Omron CX-Programmer project 新規ﾌﾟﾛｼﾞｪｸﾄ (CX-Programmer 9.61)

# PLC hoge1: CP1L L

## Program 新規ﾌﾟﾛｸﾞﾗﾑ1 (cyclic task 0)
Local symbols
I 0.00 BOOL
Q 100.00 BOOL

### Section ｾｸｼｮﾝ1

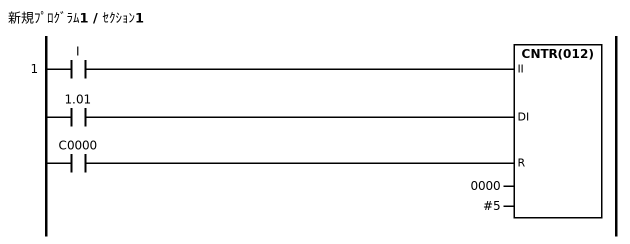
; rung 1
LD I
LD 1.01
LD C0000
CNTR(012) 0000 #5

### Section END
; rung 0
END(001)